% RSLogix 500 project ONE BUTTON CTU_BAK013.RSS, saved by version 10.00.00.00 %
PROJECT "MWL"    % processor: Bul.1763 MicroLogix 1100 Series B %

PROGRAM FILES
  LAD 2   4 rungs

DATA FILES
  O0 OUTPUT  4 elements
  I1 INPUT  6 elements
  S2 STATUS  66 elements
  B3 BINARY  2 elements
  T4 TIMER  1 elements
  C5 COUNTER  1 elements
  R6 CONTROL  1 elements
  N7 INTEGER  1 elements
  F8 FLOAT  1 elements

LADDER 2
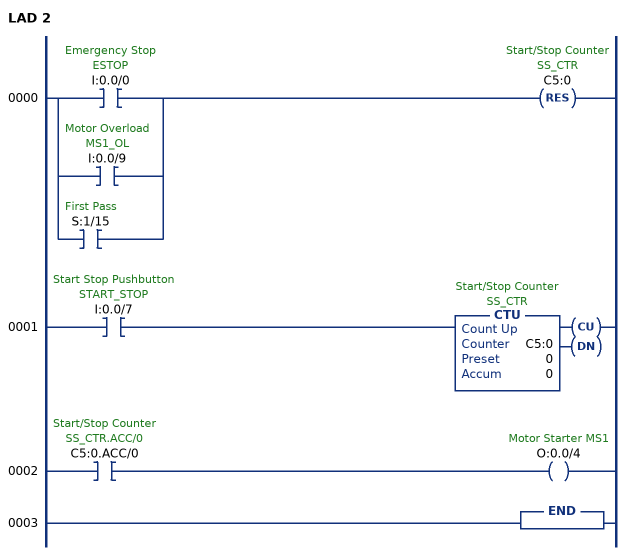
% Rung: 0 %
SOR BST XIC I:0.0/0 NXB XIC I:0.0/9 NXB XIC S:1/15 BND RES C5:0 EOR
%   I:0.0/0  ESTOP  "Emergency Stop" %
%   I:0.0/9  MS1_OL  "Motor Overload" %
%   S:1/15  "First Pass" %
%   C5:0  SS_CTR  "Start/Stop Counter" %
% Rung: 1 %
SOR XIC I:0.0/7 CTU C5:0 0 0 EOR
%   I:0.0/7  START_STOP  "Start Stop Pushbutton" %
%   C5:0  SS_CTR  "Start/Stop Counter" %
% Rung: 2 %
SOR XIC C5:0.ACC/0 OTE O:0.0/4 EOR
%   C5:0  SS_CTR  "Start/Stop Counter" %
%   O:0.0/4  MS1  "Motor Starter" %
% Rung: 3 %
SOR END EOR
